DATA_BLOCK "PilzData_fb_DB"
{ S7_Optimized_Access := 'TRUE' }
VERSION : 0.1
NON_RETAIN
"PilzData_fb"

BEGIN

END_DATA_BLOCK

